// TIA Portal V19 export
DATA_BLOCK "Coilcar_PERS"   // DB79
// stored: MemoryReserve 100
   VAR RETAIN
      PersistentValues : Struct
         Move : "SpeedMachine_Par";
      END_STRUCT;
   END_VAR
BEGIN
   PersistentValues.Move.Man.VelBwd := 5000.0;
   PersistentValues.Move.Man.VelFwdHigh := 5000.0;
   PersistentValues.Move.Man.VelFwdLow := 2000.0;
   PersistentValues.Move.Man.Acc := 500.0;
   PersistentValues.Move.Man.Dec := 500.0;
   PersistentValues.Move.Man.DelayChangeVel := T#100MS;
END_DATA_BLOCK
